// TIA Portal V19 export
VAR_GLOBAL   // PLC tag table "Analoge IW"
   "EW_LF_CM01.BN01" AT %IW128 : Int;   // Leitfähigkeit Bypass Filterpumpe CM01.BN01
   "EW_LF_CM01.BN02" AT %IW130 : Int;   // Leitfähigkeit Düsen Umwälzung CM01.BN02
   "EW_LF_CM02.BN03" AT %IW132 : Int;   // Leitfähigkeit Bypass Filterpumpe CM02.BN03
   "EW_LF_CM02.BN04" AT %IW134 : Int;   // Leitfähigkeit Düsen Umwälzung CM02.BN04
   "EW_p_CM01.BP03" AT %IW136 : Int;   // Druck Filterpumpe GP01 CM01.BP03
   "EW_p_CM01.BP04" AT %IW140 : Int;   // Druck Umwälzpumpe GP02 CM01.BP04
   "EW_p_HQ01.BP01" AT %IW138 : Int;   // Druck Beutelfiltergehäuse HQ01 HQ01.BP01
   "EW_p_CM03.BP05" AT %IW142 : Int;   // Druck Umwälzpumpe GP03 CM03.BP05
   "EW_p_CM02.BP06" AT %IW144 : Int;   // Druck Filterpumpe GP04 CM02.BP06
   "EW_p_CM02.BP07" AT %IW148 : Int;   // Druck Umwälzpumpe GP05 CM02.BP07
   "EW_p_HQ02.BP02" AT %IW146 : Int;   // Druck Beutelfiltergehäuse HQ02 HQ02.BP02
   "EW_p_CM04.BP08" AT %IW150 : Int;   // Druck Umwälzpumpe GP06 CM04.BP08
   "EW_p_CM05.BP09" AT %IW152 : Int;   // Druck Entleerung Sammeltank CM05 CM05.BP09
   EW_LW_BE AT %IW154 : Int;   // Leitwert-Wert Ablauf Be-/Entladestation WR01.BF01
   "R EW 156" AT %IW156 : Int;
   "R EW 158" AT %IW158 : Int;
   "EW_Dfl_GP01.BF01" AT %IW176 : Int;   // Durchfluss Versorgung Frischsäure GP01 GP01.BF01
   "EW_Dfl_GP02.BF02" AT %IW178 : Int;   // Durchfluss Entsorgung Altsäure GP02 GP02.BF02
   "EW_Niv_GP01.BL30" AT %IW180 : Int;   // Füllstand Versorgung Frischsäure GP01 GP01.BL30
   "EW_Niv_GP02.BL31" AT %IW182 : Int;   // Füllstand Entsorgung Altsäure GP02 GP02.BL31
   EW_WZ_rechts_1 AT %IW200 : Int;   // Hubwerk rechts Wägezelle 1 WR04.BW01
   EW_WZ_rechts_2 AT %IW202 : Int;   // Hubwerk rechts Wägezelle 2 WR04.BW02
   EW_WZ_rechts_3 AT %IW204 : Int;   // Hubwerk rechts Wägezelle 3 WR04.BW03
   EW_WZ_rechts_4 AT %IW206 : Int;   // Hubwerk rechts Wägezelle 4 WR04.BW04
   EW_WZ_links_1 AT %IW208 : Int;   // Hubwerk links Wägezelle 1 WR05.BW01
   EW_WZ_links_2 AT %IW210 : Int;   // Hubwerk links Wägezelle 2 WR05.BW02
   EW_WZ_links_3 AT %IW212 : Int;   // Hubwerk links Wägezelle 3 WR05.BW03
   EW_WZ_links_4 AT %IW214 : Int;   // Hubwerk links Wägezelle 4 WR05.BW04
   EW_Last_rechts AT %IW216 : Int;   // Hubwerk rechts Lastmessbolzen WR04.BW34
   EW_Last_links AT %IW218 : Int;   // Hubwerk links Lastmessbolzen WR05.BW43
   "R EW 220" AT %IW220 : Int;
   "R EW 222" AT %IW222 : Int;
END_VAR
